// TIA Portal V17 export
// export: Created 2024-08-09T12:53:24.4217183Z, ExportSetting WithDefaults, DisplayName Totally Integrated Automation Portal, DisplayVersion V17 Update 7, DisplayName TIA Portal Openness, DisplayVersion V17 Update 7, DisplayName TIA Portal Version Control Interface, DisplayVersion V17, DisplayName STEP 7 Professional, DisplayVersion V17 Update 7, DisplayName STEP 7 Safety, DisplayVersion V17 Update 6, DisplayName WinCC Professional, DisplayVersion V17 Update 7
TYPE "S_COMPO_FAB_ENS"
// stored: IsFailsafeCompliant false
   STRUCT
      _Incor { ExternalAccessible := 'False'; ExternalVisible := 'False'; ExternalWritable := 'False'} : String["T_CD_LINC"];   // type de composant ou lieu d'incorporation
      _CdMat { ExternalAccessible := 'False'; ExternalVisible := 'False'; ExternalWritable := 'False'} : String["T_CD_MAT"];   // code mp
      _LbMat { ExternalAccessible := 'False'; ExternalVisible := 'False'; ExternalWritable := 'False'} : String["T_LB_MAT"];   // libelle mp
      _Cel { ExternalAccessible := 'False'; ExternalVisible := 'False'; ExternalWritable := 'False'} : String["T_CD_CEL"];   // code cellule
      _Densite { ExternalAccessible := 'False'; ExternalVisible := 'False'; ExternalWritable := 'False'} : Real;   // densite produit
      _Pourcent { ExternalAccessible := 'False'; ExternalVisible := 'False'; ExternalWritable := 'False'} : Real;   // pourcentage
      _Pourcentcor { ExternalAccessible := 'False'; ExternalVisible := 'False'; ExternalWritable := 'False'} : Real;   // pourcentage corrige
      _Pcreel { ExternalAccessible := 'False'; ExternalVisible := 'False'; ExternalWritable := 'False'} : Real;   // pourcentage reel
      _Poidsreel { ExternalAccessible := 'False'; ExternalVisible := 'False'; ExternalWritable := 'False'} : Real;   // poids reel
      _TolInf { ExternalAccessible := 'False'; ExternalVisible := 'False'; ExternalWritable := 'False'} : Real;   // Tolerance poids inferieur
      _TolSup { ExternalAccessible := 'False'; ExternalVisible := 'False'; ExternalWritable := 'False'} : Real;   // Tolerance poids superieur
      _TolConfInf { ExternalAccessible := 'False'; ExternalVisible := 'False'; ExternalWritable := 'False'} : Real;   // Tolerance de non conformite inferieure
      _TolConfSup { ExternalAccessible := 'False'; ExternalVisible := 'False'; ExternalWritable := 'False'} : Real;   // Tolerance de non conformite superieure
      _Indexcel { ExternalAccessible := 'False'; ExternalVisible := 'False'; ExternalWritable := 'False'} : Int := -1;   // Index cellule en table
      _Abandon { ExternalAccessible := 'False'; ExternalVisible := 'False'; ExternalWritable := 'False'} : Bool;
   END_STRUCT;
END_TYPE
